(* PLC project Unnamed, Неизвестно Unnamed 1 *)
(* stored: creationDateTime 2024-04-05T21:53:22, modificationDateTime 2024-04-05T21:54:17 *)

PROGRAM program0
  VAR
    PID0 : PID;
  END_VAR

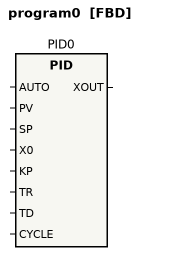
(* FBD diagram, written out as Structured Text *)
PID0();
END_PROGRAM

CONFIGURATION Config0
  RESOURCE Res0 ON PLC
    TASK task0(INTERVAL := T#20ms, PRIORITY := 0);
    PROGRAM instance0 WITH task0 : program0;
  END_RESOURCE
END_CONFIGURATION
